// TIA Portal V17 export
// export: Created 2026-04-13T11:12:44.4238455Z, ExportSetting WithDefaults, DisplayName Totally Integrated Automation Portal, DisplayVersion V17 Update 4, DisplayName TIA Portal Openness, DisplayVersion V17 Update 4, DisplayName TIA Portal Version Control Interface, DisplayVersion V17, DisplayName SINAMICS Startdrive Advanced, DisplayVersion V17, DisplayName SINAMICS Startdrive G130, G150, S120, S150, SINAMICS MV, S210, DisplayVersion V17, DisplayName SINAMICS Startdrive G110M, G120, G120C, G120D, G120P, G115D, DisplayVersion V17, DisplayName STEP 7 Professional, DisplayVersion V17 Update 4, DisplayName STEP 7 Safety, DisplayVersion V17, DisplayName WinCC Professional, DisplayVersion V17 Update 4
DATA_BLOCK "A14-阀反馈报警_DB"   // DB36
VERSION : 0.1
// stored: AutoNumber true, DBAccessibleFromOPCUA true, DBAccessibleFromWebserver true, InstanceOfName A14-阀反馈报警, InstanceOfType FB
"A14-阀反馈报警"
   // VAR
   //    补氮阀 : "A8-阀开关报警";
   //    进氮阀 : "A8-阀开关报警";
   //    泄压阀 : "A8-阀开关报警";
   //    气流雾化阀 : "A8-阀开关报警";
   //    输送进风阀 : "A8-阀开关报警";
   //    开式排风隔断阀 : "A8-阀开关报警";
   //    闭式排风隔断阀 : "A8-阀开关报警";
   //    开式进风隔断阀 : "A8-阀开关报警";
   //    闭式进风隔断阀 : "A8-阀开关报警";
   //    一级冷却水阀 : "A8-阀开关报警";
   //    二级冷冻水阀 : "A8-阀开关报警";
   //    一级排液阀 : "A8-阀开关报警";
   //    二级排液阀 : "A8-阀开关报警";
   //    除雾排液阀 : "A8-阀开关报警";
   //    溶剂回收排放阀 : "A8-阀开关报警";
   //    进风冷却水阀 : "A8-阀开关报警";
   //    塔顶清洗球阀 : "A8-阀开关报警";
   //    清洗伸缩气缸 : "A8-阀开关报警";
   //    "71阀开关报警_Instance" { S7_SetPoint := 'True'} : "A8-阀开关报警";
   //    "71阀开关报警_Instance_1" { S7_SetPoint := 'True'} : "A8-阀开关报警";
   // END_VAR
BEGIN
END_DATA_BLOCK
